Universal Robots PolyScope program: orange_Hospital_big_top.urp

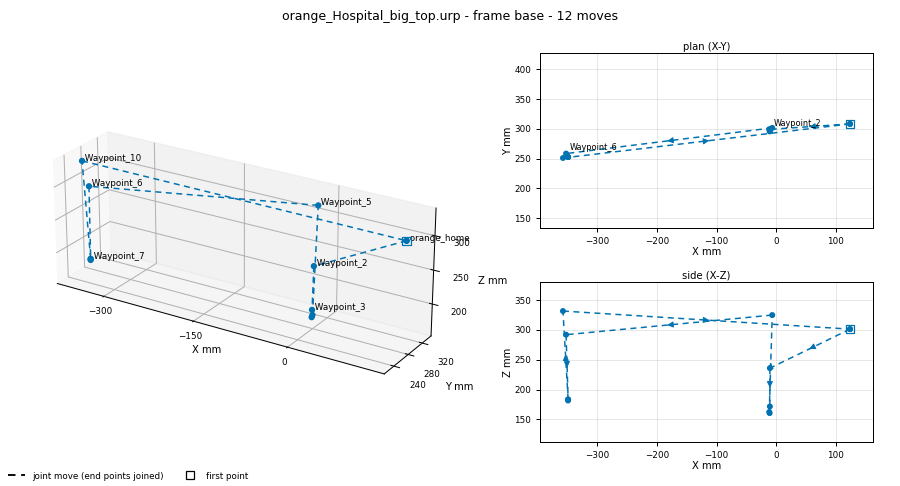
[picture p0: tool path of orange_Hospital_big_top.urp in frame base, 12 of 12 moves have a stored position in this frame; points joined in program order, loops and branches not executed]
Program orange_Hospital_big_top (installation=default directory=/programs/usbdisk/Zahra1/orangi createdIn=5.11.11.1010533 lastSavedIn=5.11.11.1010533 robotSerialNumber=20205300864)
Calibrated DH parameters: a=[-0.000166, -0.243494, -0.153108, 0.000057, -0.000123, 0]; d=[0.151897, -1.34267, 53.988124, -52.514559, 0.085283, 0.092193]; alpha=[1.572472, -0.003756, 0.002824, 1.570807, -1.572621, 0]; deltaTheta=[0, 0.020704, 7.033215, -0.770746, 0.000004, 0]
Robot Program (runOnlyOnce=true)
  MoveJ speed 60 deg/s, acceleration 80 deg/s^2 (useActiveTCP=true) feature=Base
    Waypoint orange_home: TCP in base x=124.286 y=308.277 z=301.462 mm, rx=2.2499 ry=-2.1846 rz=-0.0963 rad; joints [-269.66, -91.226, -90.279, -86.086, 92.69, 808.818] deg
    URCap Gripper (Robotiq_Grippers, Robotiq Inc.) dataModel(position=46.666666666666664, force=70.0, speed=27.0, positionInDouble=46.666666666666664, forceInDouble=70.0, speedInDouble=27.0, slaveIds=[9], blocking=true, robotCompliant=false)
    Waypoint Waypoint_2: TCP in base x=-10.32 y=299.065 z=235.916 mm, rx=2.194 ry=-2.2269 rz=-0.0307 rad; joints [-242.607, -85.6, -113.047, -70.431, 91.24, 838.401] deg
    Waypoint Waypoint_3: TCP in base x=-10.385 y=295.959 z=171.511 mm, rx=2.1851 ry=-2.2122 rz=-0.0264 rad; joints [-242.611, -93.279, -125.041, -51.182, 92.098, 838.306] deg
    Waypoint Waypoint_11: TCP in base x=-10.758 y=295.832 z=160.417 mm, rx=2.185 ry=-2.2122 rz=-0.0265 rad; joints [-242.533, -95.322, -126.662, -47.514, 92.094, 838.397] deg
    URCap Gripper (Robotiq_Grippers, Robotiq Inc.) dataModel(position=83.92156862745098, force=70.0, speed=27.0, positionInDouble=83.92156862745098, forceInDouble=70.0, speedInDouble=27.0, slaveIds=[9], blocking=true, robotCompliant=true)
    Waypoint Waypoint_4: motionParameters(jointSpeed=0.698132 jointAcceleration=0.523599 cartesianSpeed=0.25 cartesianAcceleration=1.2); TCP in base x=-11.448 y=299.206 z=162.171 mm, rx=2.1849 ry=-2.2122 rz=-0.0179 rad; joints [-242.705, -95.806, -125.307, -48.699, 92.01, 838.217] deg
    Waypoint Waypoint_5: TCP in base x=-6.395 y=301.571 z=325.057 mm, rx=2.1848 ry=-2.2122 rz=-0.0179 rad; joints [-243.819, -84.309, -89.613, -95.933, 91.999, 836.991] deg
    Waypoint Waypoint_6: TCP in base x=-352.706 y=258.458 z=292.1 mm, rx=-0.0212 ry=-3.1076 rz=-0.1101 rad; joints [-198.131, -117.528, -59.332, -90.052, 86.609, 972.629] deg
    Waypoint Waypoint_7: TCP in base x=-349.275 y=252.637 z=183.284 mm, rx=-0.035 ry=-3.0619 rz=-0.0785 rad; joints [-197.975, -120.887, -85.127, -58.714, 88.478, 973.397] deg
    Waypoint Waypoint_8: motionParameters(jointSpeed=0.523599 jointAcceleration=0.349066 cartesianSpeed=0.25 cartesianAcceleration=1.2); TCP in base x=-349.414 y=252.721 z=181.586 mm, rx=-0.0349 ry=-3.0619 rz=-0.0785 rad; joints [-197.981, -121.101, -85.28, -58.352, 88.478, 973.389] deg
    URCap Gripper (Robotiq_Grippers, Robotiq Inc.) dataModel(position=52.549019607843135, force=70.0, speed=18.0, positionInDouble=52.549019607843135, forceInDouble=70.0, speedInDouble=18.0, slaveIds=[9], blocking=true, robotCompliant=true)
    Waypoint Waypoint_7: TCP in base x=-349.275 y=252.637 z=183.284 mm, rx=-0.035 ry=-3.0619 rz=-0.0785 rad; joints [-197.975, -120.887, -85.127, -58.714, 88.478, 973.397] deg
    Waypoint Waypoint_10: TCP in base x=-357.933 y=251.051 z=331.828 mm, rx=-0.0183 ry=-3.1351 rz=-0.107 rad; joints [-196.825, -120.332, -43.412, -104.787, 86.204, 973.84] deg
    Waypoint orange_home: TCP in base x=124.286 y=308.277 z=301.462 mm, rx=2.2499 ry=-2.1846 rz=-0.0963 rad; joints [-269.66, -91.226, -90.279, -86.086, 92.69, 808.818] deg
